(* IEC 61131-3 sources: s22-soft-shell/st_interpret/tests/test_inputs/execution/st_subset_1, 10 files *)

(* ---- 01_Bool.st ---- *)
PROGRAM 01_real
    VAR
		a : bool;
        ST_TESTING_RESULT : bool;
    END_VAR
		a := TRUE;
        ST_TESTING_RESULT := (a = true);
END_PROGRAM

(* ---- 01_Bool_01.st ---- *)
PROGRAM 01_real //boolean accepts integers 0 and 1
    VAR
	a : bool;
        b : bool;
        c : bool;
        d : bool;
        ST_TESTING_RESULT : bool;
    END_VAR
	a := TRUE;
        b := FALSE;
        c := 1; //true
        d := 0; //false

        ST_TESTING_RESULT := (a & not b) & (c & not d);
END_PROGRAM

(* ---- 01_Int.st ---- *)
PROGRAM 01_Int
    VAR
		a : INT;
        ST_TESTING_RESULT : bool;
    END_VAR
		a := 1;
        ST_TESTING_RESULT := (a = 1);
END_PROGRAM

(* ---- 01_mixed.st ---- *)
PROGRAM 01_real //accepts all types in same program
    VAR
	a : real;
        b : int;
        c : bool;
        ST_TESTING_RESULT : bool;
    END_VAR
	a := 1.2;
        b := 5;
        c := True;
        ST_TESTING_RESULT := (a = 1.2) & ((b = 5) & c);
END_PROGRAM

(* ---- 01_Multi.st ---- *)
PROGRAM 01_Multi
    VAR
        a : INT;
        b : INT;
        c : INT;
        ST_TESTING_RESULT : bool;
    END_VAR
        a := 1;
        b := 2;
        c := 3;
        ST_TESTING_RESULT := ((a = 1) & (b = 2)) & (c = 3);
END_PROGRAM

(* ---- 01_NestedBool.st ---- *)
PROGRAM 01_NestedBool
    VAR
	a : bool;
        b : bool;
        c : bool;
        ST_TESTING_RESULT : bool;
    END_VAR
	a := true;
        b := a;
        c := b;
        ST_TESTING_RESULT := a & (b & c);
END_PROGRAM

(* ---- 01_NestedInt.st ---- *)
PROGRAM 01_NestedInt
    VAR
	a : INT;
        b : INT;
        c : INT;
        ST_TESTING_RESULT : bool;
    END_VAR
 	a := 1;
        b := a;
        c := b;
        ST_TESTING_RESULT := ((a = 1) & (b = 1)) & (c = 1);
END_PROGRAM

(* ---- 01_NestedReal.st ---- *)
PROGRAM 01_NestedReal
    VAR
	a : real;
        b : real;
        c : real;
        ST_TESTING_RESULT : bool;
    END_VAR
	a := 1.5;
        b := a;
        c := b;
        ST_TESTING_RESULT := ((a = 1.5) & (b = 1.5)) & (c = 1.5);
END_PROGRAM

(* ---- 01_Real.st ---- *)
PROGRAM 01_real
    VAR
		a : real;
        ST_TESTING_RESULT : bool;
    END_VAR
		a := 1.2;
        ST_TESTING_RESULT := (a = 1.2);
END_PROGRAM

(* ---- 01_truncate.st ---- *)
PROGRAM 01_truncate //should not error but rather truncate 1.5 to 1
    VAR
	a : INT;
        ST_TESTING_RESULT : bool;
    END_VAR
	a := 1.5;
        ST_TESTING_RESULT := (a = 1);
END_PROGRAM
